FUNCTION_BLOCK fb_oeprationChuck
VAR_INPUT
END_VAR
VAR_OUTPUT
END_VAR
VAR
	SFCInit : bool;
	flgInitDone: BOOL;
	trn_chuckCloseDone: BOOL;
	trn_chuckOpenDone: BOOL;
END_VAR

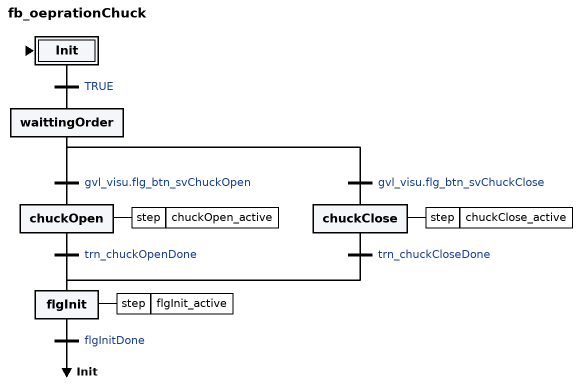
INITIAL_STEP Init:
END_STEP
TRANSITION FROM Init TO waittingOrder
    := TRUE;
END_TRANSITION
STEP waittingOrder:
END_STEP
TRANSITION FROM waittingOrder TO chuckOpen
    := gvl_visu.flg_btn_svChuckOpen;
END_TRANSITION
STEP chuckOpen:
    chuckOpen_active(N);  // step action
END_STEP
TRANSITION FROM chuckOpen TO flgInit
    := trn_chuckOpenDone;
END_TRANSITION
TRANSITION FROM waittingOrder TO chuckClose
    := gvl_visu.flg_btn_svChuckClose;
END_TRANSITION
STEP chuckClose:
    chuckClose_active(N);  // step action
END_STEP
TRANSITION FROM chuckClose TO flgInit
    := trn_chuckCloseDone;
END_TRANSITION
STEP flgInit:
    flgInit_active(N);  // step action
END_STEP
TRANSITION FROM flgInit TO Init
    := flgInitDone;
END_TRANSITION

ACTION chuckClose_active:
IF chuckClose._x AND chuckClose.x = FALSE THEN
	trn_chuckCloseDone := FALSE;
	gvl_solv.fbi_chuck.in_flg_run := FALSE;
	gvl_solv.fbi_chuck.in_var_moveMode := eP_svMoveMode.svB;
ELSIF chuckClose._x AND chuckClose.x THEN
	gvl_solv.fbi_chuck.in_flg_run := TRUE;
	IF gvl_solv.fbi_chuck.out_flg_Done THEN
		gvl_solv.fbi_chuck.in_flg_run := FALSE;
		trn_chuckCloseDone := TRUE;
	END_IF
END_IF
END_ACTION

ACTION chuckOpen_active:
IF chuckOpen._x AND chuckOpen.x = FALSE THEN
	trn_chuckOpenDone := FALSE;
	gvl_solv.fbi_chuck.in_flg_run := FALSE;
	gvl_solv.fbi_chuck.in_var_moveMode := eP_svMoveMode.svA;
ELSIF chuckOpen._x AND chuckOpen.x THEN
	gvl_solv.fbi_chuck.in_flg_run := TRUE;
	IF gvl_solv.fbi_chuck.out_flg_Done THEN
		gvl_solv.fbi_chuck.in_flg_run := FALSE;
		trn_chuckOpenDone := TRUE;
	END_IF
END_IF
END_ACTION

ACTION flgInit_active:
IF flgInit._x AND flgInit.x = FALSE THEN
	flgInitDone := FALSE;
	gvl_visu.flg_btn_svChuckOpen := FALSE;
	gvl_visu.flg_btn_svChuckClose := FALSE;
ELSIF flgInit._x AND flgInit.x THEN
	flgInitDone := TRUE;
END_IF
END_ACTION

PROPERTY p_Init : bool
GET
p_init := THIS^.SFCInit;
END_GET
SET
THIS^.SFCInit := p_Init;
END_SET
END_PROPERTY

END_FUNCTION_BLOCK

(* stored: Version 1.1.0.1, ProductVersion 3.1.4024.11
   POU fb_oeprationChuck: Id {ac387cae-92e9-49e4-9912-437ade1c70b9}, SpecialFunc None
   Action chuckClose_active: Id {09982e31-bdf3-4c81-b61a-f1304d304420}
   Action chuckOpen_active: Id {74539558-0944-47c6-81a4-61498b45be90}
   Action flgInit_active: Id {28ebd55c-d14f-4d0f-b723-f30c31855163}
   Property p_Init: Id {d65f7c1d-f5d8-446a-9aa1-4f1adc614b11}
   Get Get: Id {e657e4ca-8622-4fe6-837e-1adc6fbe6a3f}
   Set Set: Id {ed776025-e418-48a3-8275-3d3098a7ef0e} *)
